// TIA Portal V20 export
// export: Created 2026-07-16T13:01:12.9350839Z, ExportSetting WithDefaults, DisplayName Totally Integrated Automation Portal, DisplayVersion V20 Update 5, DisplayName TIA Portal Openness, DisplayVersion V20 Update 4, DisplayName TIA Portal Version Control Interface, DisplayVersion V20 Update 5, DisplayName SINAMICS Startdrive Advanced, DisplayVersion V20, DisplayName SINAMICS DCC, DisplayVersion V20, DisplayName SINAMICS Startdrive G130, G150, S120, S150, SINAMICS MV, G220, S200, S210, DisplayVersion V20, DisplayName SINAMICS Startdrive G110M, G120, G120C, G120D, G120P, G115D, DisplayVersion V20, DisplayName STEP 7 Professional, DisplayVersion V20 Update 5, DisplayName STEP 7 Safety, DisplayVersion V20 Update 2, DisplayName WinCC Basic/Comfort/Advanced, DisplayVersion V20 Update 5, DisplayName WinCC Unified, DisplayVersion V20 Update 5
TYPE "UDT_ShredderSequencerIO"
// stored: IsFailsafeCompliant false
   STRUCT
      CycleStart : Bool;
      CycleStop : Bool;
      DownstreamRunning : Bool;
      DischargeConvRunning : Bool;
      HopperLevelHigh : Bool;
      ShredderRunFwdFB : Bool;
      ShredderMotorCurrent : Real;
      MotorFaultActive : Bool;
      FaultReset : Bool;
      OperatorPusherMode : Int;
      PusherJogPreStartSounder : Bool;
      "Step" : Int;
      DischargeConveyorTimeoutFault : Bool;
      ShredderBlockedFault : Bool;
      RunDischargeConv : Bool;
      RunInfeedConv : Bool;
      EnableUpstream : Bool;
      PreStartSounder : Bool;
      InCycle : Bool;
      MotorReverseCmd : Bool;
      MotorAutoStartCmd : Bool;
      MotorPreStartDoneCmd : Bool;
      PusherModeCmd : Int;
   END_STRUCT;
END_TYPE
